{attribute 'qualified_only'}
{attribute 'strict'}
TYPE StateCnv :
(
	Off,
	Reset,
	Power,
	Ready,
	Moving
);
END_TYPE

(* stored: Version 1.1.0.1, ProductVersion 3.1.4024.3
   DUT StateCnv: Id {6e2083ee-cb86-49d0-b796-c53ec180a773} *)
